Fanuc KAREL source: ko00011.KL

-- PROVISIONAL review KL for V940-1; original PC SHA256 54e67a8545f01739322a8c2a21a08198870f63ff0b9da430ca6be9e6a12fb5a3
-- Incomplete behavior may be omitted. Consult companion uncertainty JSON. Do not deploy.
PROGRAM KO00011
%NOLOCKGROUP
-- UNRESOLVED_DECL P1 type=000102
-- UNRESOLVED_DECL P2 type=000102
-- UNRESOLVED_DECL P3 type=000102
-- UNRESOLVED_DECL OUT type=000106
BEGIN
  -- V9_ZERO_TABLE_METADATA_HINT layout=0001; no indexed target words; source/name/runtime held
  -- UNRESOLVED_PC offsets 5-65; opcodes 27,27,49,7E,AD,27,49,7E,AD,27,49,7E,AD,76,7E,4A
  -- UNRESOLVED_PC offsets 70-74; opcodes 7F
END KO00011
